FUNCTION_BLOCK VECTOR_GET_ANGLE (* Gets angle between two vectors *)
  (* Standard: 61499-2 *)
  (* Version 1.0, 02-05-12, GASR, Universidade do Estado de Santa Catarina *)
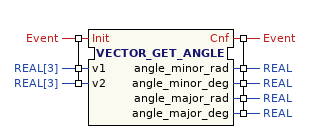
  EVENT_INPUT
    Init WITH v1, v2;
  END_EVENT
  EVENT_OUTPUT
    Cnf WITH angle_minor_rad, angle_minor_deg, angle_major_rad, angle_major_deg;
  END_EVENT
  VAR_INPUT
    v1 : ARRAY [0..2] OF REAL;
    v2 : ARRAY [0..2] OF REAL;
  END_VAR
  VAR_OUTPUT
    angle_minor_rad : REAL;
    angle_minor_deg : REAL;
    angle_major_rad : REAL;
    angle_major_deg : REAL;
  END_VAR
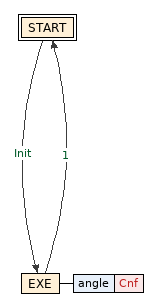
  EC_STATES
    START;
    EXE : angle -> Cnf;
  END_STATES
  EC_TRANSITIONS
    START TO EXE := Init;
    EXE TO START := 1;
  END_TRANSITIONS
  ALGORITHM angle IN Lua:
local v1_abs = ( ( v1[ 1 ]^2 ) + ( v1[ 2 ]^2 ) + ( v1[ 3 ]^2 ) )^0.5
local v2_abs = ( ( v2[ 1 ]^2 ) + ( v2[ 2 ]^2 ) + ( v2[ 3 ]^2 ) )^0.5
angle_minor_rad = 0
for i = 1, 3 do
        angle_minor_rad = angle_minor_rad + v1[ i ]*v2[ i ]
end
angle_minor_rad = ( angle_minor_rad/( v1_abs*v2_abs ) )
angle_minor_rad = math.acos( angle_minor_rad )
angle_major_rad = (2*math.pi) - angle_minor_rad
angle_minor_deg = (( angle_minor_rad*360 )/( 2*math.pi ) )
angle_major_deg = 360 - angle_minor_deg
  END_ALGORITHM
END_FUNCTION_BLOCK
